FUNCTION F_denormalization : LREAL
VAR_INPUT
	x : LREAL;
	mean : LREAL;
	std : LREAL;
END_VAR

F_denormalization := x * std + mean;

END_FUNCTION

(* stored: Version 1.1.0.1, ProductVersion 3.1.4024.12
   POU F_denormalization: Id {86002d00-668b-43f5-be54-085674f22bae}, SpecialFunc None *)
